INTERFACE PUBLIC CompletingCommands

METHOD PUBLIC Abort
END_METHOD

METHOD PUBLIC StateComplete
END_METHOD

METHOD PUBLIC Stop
END_METHOD

END_INTERFACE

(* stored: Version 1.1.0.1, ProductVersion 3.1.4026.12
   Itf CompletingCommands: Id {81f78d50-be70-0fcb-055f-f4ffcddca7b0}
   Method Abort: Id {8ee5afdd-51e7-4fa3-a57e-ea76fca8a760}
   Method StateComplete: Id {099e1bb1-b80d-43a9-be21-ee099858952a}
   Method Stop: Id {e742b291-4d90-44a0-afd4-1eae1c0474c0} *)
